Fanuc KAREL source: inv_only.kl

PROGRAM INV_ONLY
%INVISIBLE
VAR
	I : INTEGER
BEGIN
	I = 1
	WRITE('I = ', I, CR)
END INV_ONLY
